FUNCTION_BLOCK FB_CTU_UDINT (* counters (up-counter) *)
  (* Standard: 61131-3; Classification: counters *)
  (* Version 1.0, 2009-09-14, 4DIAC-IDE, 4DIAC-Consortium *)
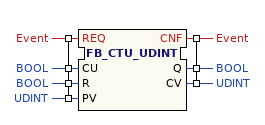
  EVENT_INPUT
    REQ WITH CU, PV, R; (* Service Request *)
  END_EVENT
  EVENT_OUTPUT
    CNF WITH Q, CV; (* Confirmation of Requested Service *)
  END_EVENT
  VAR_INPUT
    CU : BOOL; (* Count up (Rising Edge Detection) *)
    R : BOOL; (* Reset *)
    PV : UDINT; (* Preset value *)
  END_VAR
  VAR_OUTPUT
    Q : BOOL; (* Output *)
    CV : UDINT; (* Count value *)
  END_VAR
  (* Service APPLICATION/RESOURCE: counters (up-counter) *)
END_FUNCTION_BLOCK
